{attribute 'GeneratedUsingTerminal: EK1100-0000-0018'}
{attribute addProperty BoxType "EK1100-0000-0018"}
{attribute addProperty Id "RC60_A2_EK1122RC60_A2_EK1122_620268C073RC60_A3_EK1122RC60_A3_EK1122_0BEA55B5120RC60_A5_EL1809EL1809_32157CFD20RC60_A6_EL1809EL1809_32157CFD20RC60_A7_EL2809EL2809_2B6483BD19RC60_A8_EL2809EL2809_2B6483BD19RC60_A9_EL2809EL2809_2B6483BD19RC60_1_EndTerminal_EL9010EL9010_D29C20850"}
{attribute addProperty CRC "2611717856"}
{attribute addProperty Size "290"}
{attribute addProperty Name "RC60_1 (EK1100)"}
TYPE RC60_1_EK1100_9BABA6E0 EXTENDS EK1100_1FC0878B :
STRUCT
	{attribute addProperty Name "RC60_A2 (EK1122)"}
	{attribute addProperty PreviousPort "RC60_1 (EK1100) : B"}
	RC60_A2_EK1122 : RC60_A2_EK1122_620268C0;
	{attribute addProperty Name "RC60_A3 (EK1122)"}
	{attribute addProperty PreviousPort "RC60_A2 (EK1122) : C"}
	RC60_A3_EK1122 : RC60_A3_EK1122_0BEA55B5;
	{attribute addProperty Name "RC60_A5 (EL1809)"}
	{attribute addProperty PreviousPort "RC60_A3 (EK1122) : C"}
	RC60_A5_EL1809 : EL1809_32157CFD;
	{attribute addProperty Name "RC60_A6 (EL1809)"}
	{attribute addProperty PreviousPort "RC60_A5 (EL1809) : B"}
	RC60_A6_EL1809 : EL1809_32157CFD;
	{attribute addProperty Name "RC60_A7 (EL2809)"}
	{attribute addProperty PreviousPort "RC60_A6 (EL1809) : B"}
	RC60_A7_EL2809 : EL2809_2B6483BD;
	{attribute addProperty Name "RC60_A8 (EL2809)"}
	{attribute addProperty PreviousPort "RC60_A7 (EL2809) : B"}
	RC60_A8_EL2809 : EL2809_2B6483BD;
	{attribute addProperty Name "RC60_A9 (EL2809)"}
	{attribute addProperty PreviousPort "RC60_A8 (EL2809) : B"}
	RC60_A9_EL2809 : EL2809_2B6483BD;
	{attribute addProperty Name "RC60_1_EndTerminal (EL9010)"}
	{attribute addProperty PreviousPort "RC60_A9 (EL2809) : B"}
	RC60_1_EndTerminal_EL9010 : EL9010_D29C2085;
END_STRUCT
END_TYPE

(* stored: Version 1.2.0.0, ProductVersion 3.1.4024.11
   DUT RC60_1_EK1100_9BABA6E0: Id {e5705358-d957-0074-0315-904ab9332c0f} *)
